FUNCTION_BLOCK TcAxis_DMC_Tc3_Direct_Motion_Control IMPLEMENTS itfAxis
//VAR_INPUT
//END_VAR
//VAR_OUTPUT
//END_VAR
VAR
END_VAR

END_FUNCTION_BLOCK

(* stored: Version 1.1.0.1, ProductVersion 3.1.4024.11
   POU TcAxis_DMC_Tc3_Direct_Motion_Control: Id {3ecf364f-113f-4c6b-b875-0e5527cca083}, SpecialFunc None *)
